PROGRAM HMI
VAR
	eChargerType : E_ChargerType;
	

	LongestChargeTIME		: REAL;
	LastTimeShotLog			: BOOL;
	
	i : INT := 1;
END_VAR

// if clear all faults, reset abort status
IF HMI_DB.ClearFaultPB = TRUE THEN
	Trips_DB.ChargedTimerRunout := FALSE;
	Trips_DB.ChargingTimerRunout := FALSE;
	Trips_DB.DumpTimerRunout := FALSE;
	Trips_DB.ChargerSummaryFault := FALSE;
	Trips_DB.ShortingSystemUnknown := FALSE;
END_IF

IF Trips_DB.ChargedTimerRunout = TRUE OR 
	Trips_DB.ChargingTimerRunout = TRUE //OR 
	//Trips_DB.DumpTimerRunout = TRUE 
	THEN
		Trips_DB.TimerRunOutON := TRUE; 
		ELSE
			Trips_DB.TimerRunOutON := FALSE;
		END_IF
		
FOR i := 1 TO 6 BY 1 DO 
	MCP_IO.Charger[i].ChargerType := Setpoints.TDKLoad[i].eChargerType := HMI_DB.TDKLoad[i].eChargerType;
		
	IF MCP_IO.Charger[i].ChargerType = E_ChargerType.TDK12kV THEN 
		HMI_DB.TDKLoad[i].PSratedV := 12;
		ELSIF MCP_IO.Charger[i].ChargerType = E_ChargerType.TDK30kV THEN
			HMI_DB.TDKLoad[i].PSratedV := 30;
		ELSIF MCP_IO.Charger[i].ChargerType = E_ChargerType.TDK50kV THEN
			HMI_DB.TDKLoad[i].PSratedV := 50;
	END_IF
END_FOR;

IF i > 6 THEN 
	i := 1;
END_IF

END_PROGRAM

(* stored: Version 1.1.0.1, ProductVersion 3.1.4024.11
   POU HMI: Id {dcabf1a6-3ca3-40de-943d-43b2e4fd41d0}, SpecialFunc None *)
